{attribute addProperty BoxType "EL6201-0000-0018"}
{attribute addProperty Id "Configuration_okayAT %I*BOOL811Power_FailAT %I*BOOL812Auto_addresing_mode_enabledAT %I*BOOL813Auto_addressing_mode_availableAT %I*BOOL814Protected_mode_activeAT %I*BOOL815Slave_with_address_0_foundAT %I*BOOL816Offline_ReadyAT %I*BOOL817Normal_OperationAT %I*BOOL818ASI_phaseAT %I*BYTE819Power24_Mode_EnabledAT %I*BOOL8112Power24_FailAT %I*BOOL8113M4_Profile_Support_EnabledAT %I*BOOL8114TxPDO_ToggleAT %I*BOOL8116"}
{attribute addProperty CRC "287849958"}
{attribute addProperty SizeInBites "104"}
{attribute addProperty SizeInBytes "13"}
TYPE ASI_Status_11283DE6 :
STRUCT
	{attribute addProperty Name "Configuration_okay"}
	Configuration_okay AT %I* : BOOL;
	{attribute addProperty Name "Power_Fail"}
	Power_Fail AT %I* : BOOL;
	{attribute addProperty Name "Auto_addresing_mode_enabled"}
	Auto_addresing_mode_enabled AT %I* : BOOL;
	{attribute addProperty Name "Auto_addressing_mode_available"}
	Auto_addressing_mode_available AT %I* : BOOL;
	{attribute addProperty Name "Protected_mode_active"}
	Protected_mode_active AT %I* : BOOL;
	{attribute addProperty Name "Slave_with_address_0_found"}
	Slave_with_address_0_found AT %I* : BOOL;
	{attribute addProperty Name "Offline_Ready"}
	Offline_Ready AT %I* : BOOL;
	{attribute addProperty Name "Normal_Operation"}
	Normal_Operation AT %I* : BOOL;
	{attribute addProperty Name "ASI_phase"}
	ASI_phase AT %I* : BYTE;
	{attribute addProperty Name "Power24_Mode_Enabled"}
	Power24_Mode_Enabled AT %I* : BOOL;
	{attribute addProperty Name "Power24_Fail"}
	Power24_Fail AT %I* : BOOL;
	{attribute addProperty Name "M4_Profile_Support_Enabled"}
	M4_Profile_Support_Enabled AT %I* : BOOL;
	{attribute addProperty Name "TxPDO_Toggle"}
	TxPDO_Toggle AT %I* : BOOL;
END_STRUCT
END_TYPE

(* stored: Version 1.2.0.0, ProductVersion 3.1.4024.9
   DUT ASI_Status_11283DE6: Id {90b61c6c-38de-4dae-b5ee-6b91d7d5cb0d} *)
